FUNCTION_BLOCK MasterSlave (* Composite Function Block Type *)
  (* Standard: 61499-2 *)
  (* Version 0.0, 2011-03-19, Majid Sorouri, nxtControl GmbH, template *)
  (* Compiler header: package fb.rt.pnp; *)
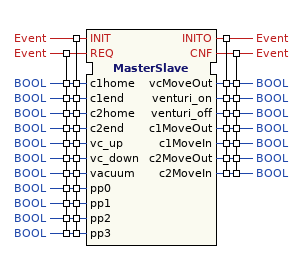
  EVENT_INPUT
    INIT WITH c1home, c1end, c2home, c2end, vc_up, vc_down, vacuum, pp0, pp1, pp2, pp3; (* Initialization Request *)
    REQ WITH c1home, c1end, c2home, c2end, vc_up, vc_down, vacuum, pp0, pp1, pp2, pp3; (* Normal Execution Request *)
  END_EVENT
  EVENT_OUTPUT
    INITO WITH venturi_off, vcMoveOut, venturi_on, c1MoveOut, c1MoveIn, c2MoveOut, c2MoveIn; (* Initialization Confirm *)
    CNF WITH vcMoveOut, venturi_on, venturi_off, c1MoveOut, c1MoveIn, c2MoveOut, c2MoveIn; (* Execution Confirmation *)
  END_EVENT
  VAR_INPUT
    c1home : BOOL;
    c1end : BOOL;
    c2home : BOOL;
    c2end : BOOL;
    vc_up : BOOL;
    vc_down : BOOL;
    vacuum : BOOL;
    pp0 : BOOL;
    pp1 : BOOL;
    pp2 : BOOL;
    pp3 : BOOL;
  END_VAR
  VAR_OUTPUT
    vcMoveOut : BOOL;
    venturi_on : BOOL;
    venturi_off : BOOL;
    c1MoveOut : BOOL;
    c1MoveIn : BOOL;
    c2MoveOut : BOOL;
    c2MoveIn : BOOL;
  END_VAR
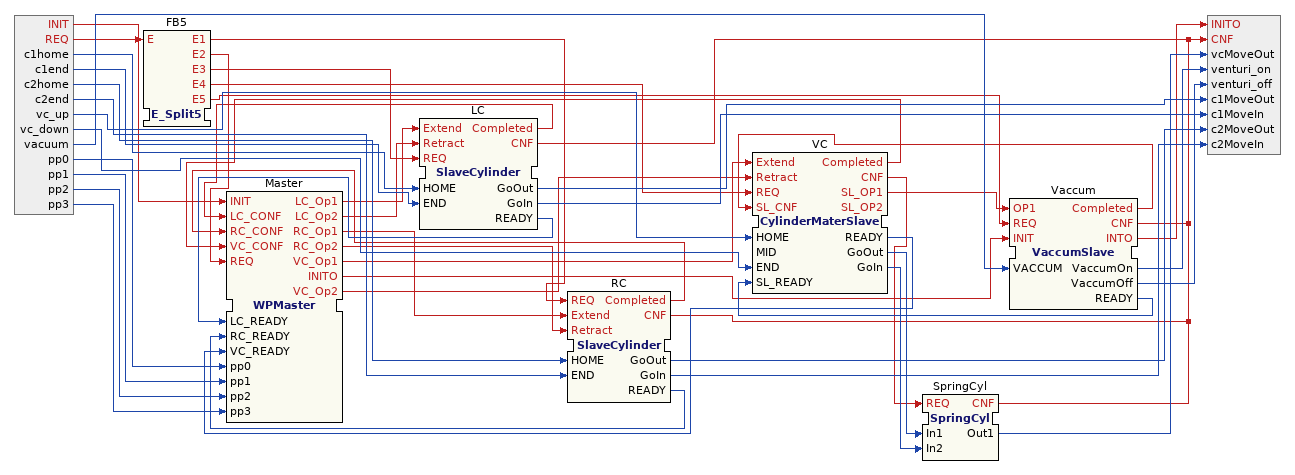
  FBS
    Vaccum : VaccumSlave;
    FB5 : E_Split5;
    LC : SlaveCylinder;
    RC : SlaveCylinder;
    VC : CylinderMaterSlave;
    Master : WPMaster;
    SpringCyl : SpringCyl;
  END_FBS
  EVENT_CONNECTIONS
    REQ TO FB5.E;
    INIT TO Master.INIT;
    FB5.E1 TO RC.REQ;
    Master.LC_Op1 TO LC.Extend;
    Master.LC_Op2 TO LC.Retract;
    Master.RC_Op1 TO RC.Extend;
    Master.RC_Op2 TO RC.Retract;
    Master.VC_Op1 TO VC.Extend;
    LC.Completed TO Master.LC_CONF;
    RC.Completed TO Master.RC_CONF;
    VC.Completed TO Master.VC_CONF;
    LC.CNF TO CNF;
    RC.CNF TO CNF;
    VC.SL_OP1 TO Vaccum.OP1;
    FB5.E2 TO Master.REQ;
    FB5.E3 TO LC.REQ;
    FB5.E4 TO VC.REQ;
    FB5.E5 TO Vaccum.REQ;
    Vaccum.Completed TO VC.SL_CNF;
    Vaccum.CNF TO CNF;
    Master.INITO TO Vaccum.INIT;
    Vaccum.INTO TO INITO;
    SpringCyl.CNF TO CNF;
    VC.CNF TO SpringCyl.REQ;
    Master.VC_Op2 TO VC.Retract;
  END_CONNECTIONS
  DATA_CONNECTIONS
    c1home TO LC.HOME;
    c1end TO LC.END;
    c2home TO RC.HOME;
    c2end TO RC.END;
    RC.GoOut TO c2MoveOut;
    RC.GoIn TO c2MoveIn;
    LC.GoOut TO c1MoveOut;
    LC.GoIn TO c1MoveIn;
    LC.READY TO Master.LC_READY;
    RC.READY TO Master.RC_READY;
    VC.READY TO Master.VC_READY;
    pp0 TO Master.pp0;
    pp1 TO Master.pp1;
    pp2 TO Master.pp2;
    pp3 TO Master.pp3;
    vc_up TO VC.HOME;
    vc_down TO VC.END;
    Vaccum.VaccumOn TO venturi_on;
    Vaccum.VaccumOff TO venturi_off;
    Vaccum.READY TO VC.SL_READY;
    VC.GoOut TO SpringCyl.In1;
    VC.GoIn TO SpringCyl.In2;
    SpringCyl.Out1 TO vcMoveOut;
    vacuum TO Vaccum.VACCUM;
  END_CONNECTIONS
END_FUNCTION_BLOCK
